PROGRAM MAIN_Fast
VAR
	Router														: FB_Teltonika;
	SystemControl												: FB_SystemControl;
	AcDcCharger													: FB_AcDcCharger;
	ACswitchgear												: FB_ACSwitchgear;
	DCLink														: FB_DCLink;
	HartingIO													: FB_HartingIO;
	NeutralTransformer											: FB_NeutralTransformer;
	Coolingsystem												: FB_Coolingsystem;
	PowerStack													: FB_PowerStack;
	PowerMonitor												: FB_PowerQualityMonitoring;
	InternalPowerSupply											: FB_InternalPowerSupply;
	BMS															: FB_BMS;
	ProtectionSystems											: FB_ProtectionSystems;
	Enclosure													: FB_enclosure;
	PLCstate													: FB_PLCState;
	Peakshavebox												: FB_peakshavebox;
	GenComm														: FB_GenComm;				
END_VAR

VAR // structures containing all system control/monitoring vars and are exchanged with other task.
	{ attribute 'TcHmiSymbol.Hide' }
	monitor						: ST_System_Monitor;
	{ attribute 'TcHmiSymbol.Hide' }
	control						: REFERENCE TO ST_System_Control;

	fb_WritePersistentData		: WritePersistentData;
END_VAR

VAR
	//Reset function
	b_ResetManual			: BOOL;
	ton_EMstopTimeOut		: TON := (PT:= T#30S);
	w_MethodFbs				: WORD;
	tp_ResetDuration		: TP := (PT:= T#2S);
	ton_ForceShutdown		: ton := (PT := T#10S);
	ton_shutdownDelay		: ton := (PT := T#3S);
	b_shutdownInitiated		: BOOL;
	ton_NUCshutdownDelay	: ton := (PT := T#20S);
	
	//Method feedbacks
	EMstopFb				: BYTE;		
	b_EMstopCompleted		: BOOL;
	b_shutdownCompleted		: BOOL;
	b_MethodStartFB			: BOOL;
	r_trigInitialReset		: R_TRIG;
END_VAR

control REF= MAIN_Slow.control;

WearLogging();
SetConfig();
SetSystemMonitorControlvars();

IF __ISVALIDREF(control) AND InitMachine() THEN
	PLCstate();
	
	Safety(b_extEmstopTrigger := SystemControl.toSystem.control.b_EMStop,
		b_enable := GVL.b_SystemReady
		);
		Safety.EDMSignals.b_NetcontactorEDM := Powerstack.b_NetcontEDM;
		Safety.EDMSignals.b_MccbMasterEDM:= Powerstack.b_MasterMccbEDM;
		Safety.EDMSignals.b_MccbSlaveEDM:= Powerstack.b_SlaveMccbEDM;
		
	//call FB
	
	PowerStack(
			e_ACRotationStateExt			:= powermonitor.get.OutputField.e_ACrotationStatus,
			r_PLossInternal					:= 0,
			r_QLossInternal					:= 0,
			st_params						:= settings.MachineParams.Powerstack,
			st_service						:= service.Powerstack,
			st_calibration 					:= settings.Calibration.Powerstack,
			set								:= SystemControl.toSystem.Powerstack,
			b_transportMode					:= systemcontrol.toSystem.b_TransportMode,
			b_DoublePowermodule				:= settings.Configuration.b_DoublePowerModule,
			b_BatteryDCReady				:= BMS.PowerStatus = eHVDC_Powerstatus.ON,
			r_BatteryDCvoltage				:= BMS.get.MBMU.BatteryStatus.r_SystemVoltage,
			b_RotationswitchEnable			:= settings.Configuration.b_AutomaticACrotation,
			b_ExtgridCodeTrip				:= Powermonitor.get.OutputField.r_CurrentUnbalance > settings.GridParams.r_CurrentUnbalanceLimit AND Powermonitor.get.OutputField.ar_Current[0] > 20 AND NOT settings.Configuration.b_NeutralTransformer,
			b_EnableFan						:= coolingsystem.b_FanPowerstackEnable,
			b_OutputConnected				:= ACswitchgear.get.b_OutputMCCBfb,
			b_InputConnected				:= ACswitchgear.get.b_inputMCCBfb,// AND ACswitchgear.get.b_InputContactorfb
			b_InternalACRequired			:= InternalPowerSupply.b_PowerStackACRequired
		);

	PowerMonitor(
		b_enable:= TRUE,
		powerstackGet := powerstack.get,
		b_TNModeActive:= Monitor.protections.Insulation.e_EarthingSystemDetected <> eEarthingsystems.IT,
		b_thirdOutputfieldAvailable := settings.Configuration.b_ThirdOutputConnection,
		b_NeutralTransformerAvailable := settings.Configuration.b_NeutralTransformer,
		b_InputFieldsAvailable := settings.Configuration.b_ACInputConnection
		);
	
	InternalPowerSupply(
			st_PowerstackDemandSupply 	:= Powerstack.st_InternalPsuSupplyRequest, 
			st_CoolingDemandSupply 		:= Coolingsystem.IPSRequest,
			st_ACDCchargerDemandSupply 	:= ACDCCharger.IPSRequest,
			st_DCBusDemandSupply		:=	dclink.st_PowerDemand,
			b_BusbarACAvailable := powerstack.get.b_ACdetected,
			st_params:=Settings.MachineParams.Interpowersupply,
			e_BMSPowerState := BMS.PowerStatus,
			b_ConditioningOnBatteryAllowed := BMS.b_InternalHVDCAllowed
		);

	BMS(
		st_params 		:= settings.MachineParams.BMS,
		st_service		:= service.BMS,
		b_HVDCEnable	:= Internalpowersupply.b_HVDC_Enable,
		set 			:= Systemcontrol.toSystem.BMS,
		by_NoOfStrings	:= Settings.Configuration.by_NoBatteryStrings
	);	

	Enclosure(st_params := Settings.MachineParams.Enclosure, set := SystemControl.toSystem.Enclosure);
		Enclosure.ledstrip.SetMachineStatus(
			b_Error := GVL.b_QuickshutdownActive OR GVL.b_EmergencyShutdownActive OR GVL.b_NormalShutdownActive,
			b_warning := GVL.b_WarningActive,
			b_attention := NOT BMS.get.BatteryInfo.b_chargingAllowed OR NOT BMS.get.BatteryInfo.b_dischargingAllowed,
			b_Normal := BMS.PowerStatus = eHVDC_powerstatus.ON,
			b_off :=  Monitor.system.e_State = eSystemState.Transport,
			r_Soc := BMS.get.BatteryInfo.r_SOCScaled,
			r_DCcurrent := Powerstack.get.r_DCcurrent);

	CoolingSystem(
		st_params := settings.MachineParams.Coolingsystem,
		InverterConditioningRequirement := powerstack.ConditioningRequirement,
		b_HVDC_Available	:=	InternalPowerSupply.Get.b_HVDCAvailable,
		b_400V_Available  := 	InternalPowerSupply.Get.b_400VACAvailable,
		
// 		by_PSsetCooling:= powerstack.by_CoolingControl,
// 		b_InverterRunning:= powerstack.get.b_InverterRunning,
// 		r_InverterLoad := powerstack.get.r_LoadPercent,
// 		b_24v_Available := internalpowersupply.Get.b_24VdcAvailable,
// 		b_400v_Available := internalpowersupply.Get.b_400VACAvailable,
// 		e_400vSupplySource := internalpowersupply.Get.e_400VSupplySource,
// 		r_BMSAverageBattTemp := BMS.get.BatteryInfo.ar_CellTemperature[eSubvalues.Average],
// 		r_BMSMaxBattTemp := BMS.get.BatteryInfo.ar_CellTemperature[eSubvalues.Maximum],
// 		b_DehumStart := systemcontrol.toSystem.control.b_startDeHum,
// 		r_enclosureHumidity := enclosure.get.climate.r_Humidity,
// 		r_enclosureTemperature := enclosure.get.climate.r_Temperature,
// 		r_InverterTemp := Powerstack.get.PowermoduleMaster.r_TemperatureInverter,
// 		b_ConditioningOnBatteryAllowed := BMS.b_InternalHVDCAllowed
		);
		
	
	NeutralTransformer(
		b_enable:= settings.Configuration.b_NeutralTransformer,
		r_currentN := Powermonitor.get.inverter.ar_Current[phases.N],
		r_linevoltage := powermonitor.get.OutputField.ar_LineVoltage[Phases.AVG],
		r_voltageUnbalance := Powermonitor.get.Outputfield.r_VoltageUnbalance,
		b_NetcontactorFB := Powerstack.get.Netcontactor.b_NetConFb,
		st_params := settings.MachineParams.NeutralTransformer
		);
	
		
	ProtectionSystems(
		st_params := settings.MachineParams.Protections,
		powermonitor := Powermonitor.get,
		b_batteryAlarm := BMS.get.Events.b_OVER_TEMP_ALARM
	);
		ProtectionSystems.ToInsuMon.b_MccbfbMaster := Powerstack.get.PowermoduleMaster.b_MccbFb;
		ProtectionSystems.ToInsuMon.b_MccbfbSlave := Powerstack.get.PowermoduleSlave.b_MccbFb;
		ProtectionSystems.ToInsuMon.b_NetContFB := Powerstack.get.Netcontactor.b_NetConFb;
		ProtectionSystems.ToInsuMon.b_ACdetected := Powerstack.get.b_ACdetected;
		ProtectionSystems.ToInsuMon.b_PENlinkFB := AcSwitchgear.get.b_PENlinkfb;
		ProtectionSystems.set := systemcontrol.toSystem.Protections;
		
	ACswitchgear(
		b_inputAvailable:= settings.Configuration.b_ACInputConnection,
		b_NeutralTransformerAvailable := settings.Configuration.b_NeutralTransformer, 
		b_MCCBinputShuntTrip := protectionsystems.get.OvercurrentProtection.b_InputAlarm,
		b_MCCBOutputShuntTrip:= protectionsystems.get.overcurrentprotection.b_OutputAlarm,
		b_TransportMode := Monitor.system.e_State = eSystemState.Transport,
		set := Systemcontrol.toSystem.ACSwitchgear,
		st_params := settings.MachineParams.ACswitchgear,
		);
		
	AcDcCharger(
		st_service := service.ACDCCharger,
		st_params := settings.MachineParams.ACDCCharger,
		enable:= Settings.Configuration.b_DcCharger,
		set := systemcontrol.tosystem.AcDcCharger,(*BMS := BMS.get.BatteryInfo,*) 
		r_Soc := BMS.get.BatteryInfo.r_SOCScaled, 
		r_SystemVoltage := BMS.get.BatteryInfo.r_SystemVoltage,
		r_SystemCurrent := BMS.get.BatteryInfo.r_SystemCurrent,
		r_MaxChargeCurrent := BMS.get.BatteryInfo.r_MaxChargeCurrentAllowed,
		b_BatteryOn := (BMS.get.BatteryInfo.e_BMS_PowerOnStatus = ePowerOnSTatus.On), 
		b_BatteryFullyCharged := (BMS.get.BatteryInfo.e_BMS_Status = eBMS_status.FullCharge)
		);
	
	DcLink(
		st_params := settings.MachineParams.DC,
		r_InvCurrentDC := Powerstack.get.r_DCcurrent,
		r_battCurrent := BMS.get.BatteryInfo.r_SystemCurrent,
		r_DCbusVoltage := BMS.get.BatteryInfo.r_SystemVoltage,
		r_BattCCL := BMS.get.BatteryInfo.r_MaxChargeCurrentAllowed,
		r_BattDCL := BMS.get.BatteryInfo.r_MaxDischargeCurrentAllowed,
		b_DCsafetyOK := safety.get.b_SafetyDCOK,
		set := systemcontrol.toSystem.DCLink	
		);
	
	HartingIO(
		st_params := settings.MachineParams.HartingIO,
		set := systemcontrol.toSystem.HartingIO,
		SystemOperating := Powerstack.get.b_StartedState,
		SystemEmStop := Monitor.system.e_State = eSystemState.EMstop,
		);
		
	GenComm(
		st_params := settings.MachineParams.GenComm,
		set := systemcontrol.toSystem.GenComm);
	
	//external measurement box (PSB)	
	Peakshavebox(st_params := settings.MachineParams.PSB,
		b_enable:= settings.Configuration.b_PeakshaverBoxEnable AND Control.SoftSettings.setup.b_PeakshaveBoxEnable);
	PeakshaveBox.set := systemcontrol.toSystem.Peakshavebox;

	
	//Router --> GPS, 4G, SMS etc.
	Router(
		st_service := service.Router,
		s_message := errorhandling.a_SMSEventBuffer, 
		st_params := Settings.MachineParams.Router,
		s_SerialNumber := settings.Properties.s_SerialNumber
	);
	monitor.system.b_SMSnumberConfigured := Router.SetSMSNumber(control.SoftSettings.system.s_SMSnumber);
	monitor.system.b_CustomNameConfigured:= Router.SetDevName(control.SoftSettings.system.s_SystemName);

	//FB with connection from user to system vars
	SystemControl(
		st_params := settings.MachineParams.system,
		st_calibration := settings.Calibration,
		monitor:= monitor, control:= control);
	

//CALL MAIN FUNCTIONS
	Reset(SystemControl.toSystem.control.b_Reset, NOT GVL.b_SystemReady OR settings.MachineParams.system.b_VDLReset);
	MainSFC();
	//System shutdown --> manually or by firesystem
	SystemShutdown(Systemcontrol.toSystem.control.b_SystemShutdown OR ProtectionSystems.b_SystemShutdownCMD);
END_IF

ACTION _aErrorSequence_entry:
SFCReset := TRUE;
END_ACTION

ACTION _aInit_active:
//INIT state
b_EMstopCompleted :=  FALSE;
Monitor.system.e_State:= eSystemState.Init;
END_ACTION

ACTION _aStandBy_active:
Powerstack.Standbycmd();
Internalpowersupply.HVDC_Enable();

IF systemcontrol.toSystem.b_TransportMode THEN
	// IF Coolingsystem.Shutdown() THEN  --> WHAT TO DO WITH THIS IN NEW COOLING MODULE?
		powerstack.Shutdowncmd();
	//END_IF
	AcSwitchgear.set.b_inputContactorOpen := TRUE;
	Monitor.system.e_State:= eSystemState.Transport;
ELSE
	Monitor.system.e_State:= eSystemState.Init;
	IF  coolingsystem.Get.CoolingSystemState = eCoolingSystemState.Circulating OR 
	coolingsystem.Get.CoolingSystemState = eCoolingSystemState.ActiveCooling OR
	coolingsystem.Get.CoolingSystemState = eCoolingSystemState.ActiveHeating THEN
		Monitor.system.e_State:= eSystemState.Conditioning;
	ELSE
		Monitor.system.e_State:= eSystemState.StandBy;
	END_IF
END_IF
END_ACTION

ACTION a_ContinousActions:
ErrorSFC();
END_ACTION

ACTION a_EmergencyShutdown_active:
SFCReset := TRUE;
b_EMstopCompleted := EMStop();
Monitor.system.e_State := eSystemState.EMstop;
InternalPowersupply.HVDC_disable();
END_ACTION

ACTION a_ErrorSequence_active:
// SFC IDENTIFICATION
Powerstack.Shutdowncmd();
Reset(FALSE, systemcontrol.toSystem.control.b_Reset);

IF GVL.b_EmergencyShutdownActive THEN
	InternalPowersupply.HVDC_disable();
	Monitor.system.e_State := eSystemState.EMstop;
END_IF
END_ACTION

ACTION a_ErrorSequence_exit:
//RELEASE MAINSEQUENCE AFTER ALL ERROR ARE CLEARED
Reset(FALSE, FALSE);
SFCReset := FALSE;
END_ACTION

METHOD PUBLIC CheckDCcurrent : BOOL
VAR_INPUT
	r_in			: REAL;
END_VAR
//checkcurrent is below limit.
CheckDCcurrent := (BMS.get.BatteryInfo.r_SystemCurrent < r_in AND powerstack.get.r_DCcurrent < r_in);
END_METHOD

METHOD EMstop : BOOL

VAR
	EMstopDone	: BOOL;
END_VAR
//EMstopDone := Powerstack.EMstop() AND 
//	Coolingsystem.EMSTOP() AND 
//	Internalpowersupply.EMstop() AND 
//	BMS.EMSTOP() AND 
//	systemcontrol.EMstop();
	
EMstopFb.0 := Powerstack.EMstop();
EMstopFb.1 := Coolingsystem.EMSTOP();
EMstopFb.2 := Internalpowersupply.EMstop();
EMstopFb.3 := BMS.EMSTOP();
EMstopFb.4 := systemcontrol.EMstop();
EMstopFb.5 := ACDCCharger.EMSTOP();;
EMstopFb.6 := TRUE;
EMstopFb.7 := TRUE;

EMstopDone:= EMstopFb = 255;

ton_EMstopTimeOut(IN:= NOT EMstopDone);
EMstop := EMstopDone; //OR ton_EMstopTimeOut.Q;

IF EMstopDone THEN
	EMstopFb := 0;
END_IF

//IF ton_EMstopTimeOut.Q THEN
//	InternalPowersupply.SystemShutdown(FALSE);
//END_IF
END_METHOD

ACTION ErrorSFC:
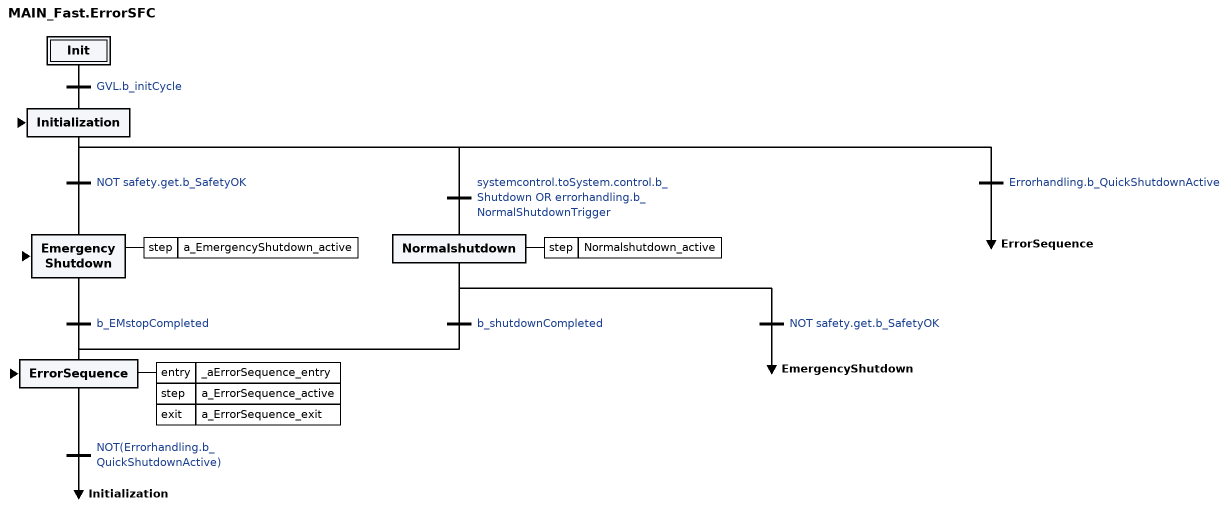
INITIAL_STEP Init:
END_STEP
TRANSITION FROM Init TO Initialization
    := GVL.b_initCycle;
END_TRANSITION
STEP Initialization:
END_STEP
TRANSITION FROM Initialization TO EmergencyShutdown
    := NOT safety.get.b_SafetyOK;
END_TRANSITION
STEP EmergencyShutdown:
    a_EmergencyShutdown_active(N);  // step action
END_STEP
TRANSITION FROM EmergencyShutdown TO ErrorSequence
    := b_EMstopCompleted;
END_TRANSITION
TRANSITION FROM Initialization TO Normalshutdown
    := systemcontrol.toSystem.control.b_Shutdown OR errorhandling.b_NormalShutdownTrigger;
END_TRANSITION
STEP Normalshutdown:
    Normalshutdown_active(N);  // step action
END_STEP
TRANSITION FROM Normalshutdown TO ErrorSequence
    := b_shutdownCompleted;
END_TRANSITION
TRANSITION FROM Normalshutdown TO EmergencyShutdown
    := NOT safety.get.b_SafetyOK;
END_TRANSITION
TRANSITION FROM Initialization TO ErrorSequence
    := Errorhandling.b_QuickShutdownActive;
END_TRANSITION
STEP ErrorSequence:  // min time T#5s
    _aErrorSequence_entry(P1);  // entry action
    a_ErrorSequence_active(N);  // step action
    a_ErrorSequence_exit(P0);  // exit action
END_STEP
TRANSITION FROM ErrorSequence TO Initialization
    := NOT(Errorhandling.b_QuickShutdownActive);
END_TRANSITION
// branch label Branch1_ErrorSFC
// branch label Branch0_ErrorSFC
END_ACTION

ACTION IdleOperation_active:
IF powerstack.stopcmd() THEN
	Monitor.system.e_State := eSystemState.Stopped;
END_IF
END_ACTION

ACTION InitializeMachine_active:

END_ACTION

METHOD PRIVATE InitMachine : Bool
VAR_INPUT
END_VAR
//Calls all available init methods of other function blocks.
//After all inits have returned true, the method returns true and main_fast operation can continue

InitMachine := TRUE;//BMS.init() AND FB.init();
END_METHOD

ACTION MainSFC:
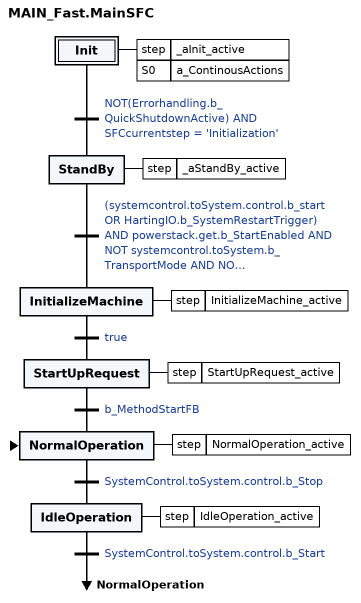
INITIAL_STEP Init:
    _aInit_active(N);  // step action
    a_ContinousActions(S0);
END_STEP
TRANSITION FROM Init TO StandBy
    := NOT(Errorhandling.b_QuickShutdownActive) AND SFCcurrentstep = 'Initialization';
END_TRANSITION
STEP StandBy:
    _aStandBy_active(N);  // step action
END_STEP
TRANSITION FROM StandBy TO InitializeMachine
    := (systemcontrol.toSystem.control.b_start OR HartingIO.b_SystemRestartTrigger) AND powerstack.get.b_StartEnabled AND NOT systemcontrol.toSystem.b_TransportMode AND NOT GVL.b_NormalShutdownActive;
END_TRANSITION
STEP InitializeMachine:
    InitializeMachine_active(N);  // step action
END_STEP
TRANSITION FROM InitializeMachine TO StartUpRequest
    := true;
END_TRANSITION
STEP StartUpRequest:
    StartUpRequest_active(N);  // step action
END_STEP
TRANSITION FROM StartUpRequest TO NormalOperation
    := b_MethodStartFB;
END_TRANSITION
STEP NormalOperation:
    NormalOperation_active(N);  // step action
END_STEP
TRANSITION FROM NormalOperation TO IdleOperation
    := SystemControl.toSystem.control.b_Stop;
END_TRANSITION
STEP IdleOperation:
    IdleOperation_active(N);  // step action
END_STEP
TRANSITION FROM IdleOperation TO NormalOperation
    := SystemControl.toSystem.control.b_Start;
END_TRANSITION
END_ACTION

ACTION NormalOperation_active:
powerstack.startcmd();

IF powerstack.get.e_State = eStatusPowerstack.running THEN
	IF NOT bms.get.BatteryInfo.b_chargingAllowed THEN
		Monitor.system.e_State := eSystemState.Discharging_Only;
	ELSIF NOT bms.get.BatteryInfo.b_DischargingAllowed THEN
		Monitor.system.e_State := eSystemState.Charging_Only;
	ELSE
		Monitor.system.e_State := eSystemState.Running;
	END_IF
ELSE
	IF powerstack.get.e_State = eStatusPowerstack.idle OR powerstack.get.e_State = eStatusPowerstack.GridCodeStop THEN
		Monitor.system.e_State := eSystemState.Stopped;	
	ELSE
		Monitor.system.e_State := eSystemState.Starting;	
	END_IF	
END_IF
END_ACTION

ACTION Normalshutdown_active:
SFCReset := TRUE;
b_shutdownCompleted := Powerstack.Shutdowncmd();
Monitor.system.e_State := eSystemState.shutdown;
END_ACTION

METHOD PUBLIC Reset : BOOL
VAR_INPUT
	b_reset	: BOOL;
	b_force : BOOL;
END_VAR
tp_ResetDuration(IN := b_reset OR b_Force);

//reinitiliaze reset statuss if reset is retriggered
IF tp_resetDuration.Q = FALSE THEN
	w_MethodFbs := 0;
END_IF


//Everything that is not automatically reset
IF tp_ResetDuration.Q AND w_MethodFbs <> 16#FF THEN
	monitor.system.e_State := eSystemState.Reset;
	
	IF NOT w_MethodFbs.0 AND b_force THEN w_MethodFbs.0 := Safety.Reset(TRUE); END_IF
	IF NOT w_MethodFbs.1 THEN w_MethodFbs.1 := InternalPowerSupply.Reset(); END_IF
	IF NOT w_MethodFbs.2 THEN w_MethodFbs.2 := Powerstack.Reset(); END_IF
	IF NOT w_MethodFbs.3 THEN w_MethodFbs.3 := protectionSystems.Reset(); END_IF
	IF NOT w_MethodFbs.4 THEN w_MethodFbs.4 := Powermonitor.Reset(); END_IF 
	IF NOT w_MethodFbs.5 THEN w_MethodFbs.5 := BMS.Reset(); END_IF 
	IF NOT w_MethodFbs.6 THEN w_MethodFbs.6 := Neutraltransformer.Reset(); END_IF
	IF NOT w_MethodFbs.7 THEN w_MethodFbs.7 := Coolingsystem.Reset(); END_IF
	IF NOT w_MethodFbs.8 THEN w_MethodFbs.8 := Router.Reset(); END_IF
	IF NOT w_MethodFbs.9 THEN w_MethodFbs.9	:= systemcontrol.Reset(); END_IF
	IF NOT w_MethodFbs.10 THEN w_MethodFbs.10:= ACDCCharger.Reset(); END_IF
	IF NOT w_MethodFbs.11 THEN w_MethodFbs.11:= TRUE; END_IF
	IF NOT w_MethodFbs.12 THEN w_MethodFbs.12:= TRUE; END_IF
	IF NOT w_MethodFbs.13 THEN w_MethodFbs.13:= TRUE; END_IF
	IF NOT w_MethodFbs.14 THEN w_MethodFbs.14:= TRUE; END_IF
	IF NOT w_MethodFbs.15 THEN w_MethodFbs.15:= TRUE; END_IF
END_IF

//Everything that is automatically reset one in error state
Reset := w_MethodFbs = 255;
END_METHOD

ACTION SetConfig:
{IF defined (ePU10_360_N_DC_IO_PSB)}
	settings.Configuration.b_PeakshaverBoxEnable 	:= TRUE;
	settings.Configuration.b_DCbuscoupling 			:= FALSE; //TRUE;
	settings.Configuration.b_NeutralTransformer		:= TRUE;
	settings.Configuration.b_ACInputConnection		:= TRUE;
	settings.Properties.s_ConfigurationCode 		:= 'ePU10_360_N_DC_IO_PSB';
{END_IF}

{IF defined (ePU10_360_N_IO_PSB)}
	settings.Properties.s_ConfigurationCode 		:= 'ePU10_360_N_IO_PSB';
	settings.Configuration.b_ACInputConnection		:= TRUE;
	settings.Configuration.b_NeutralTransformer		:= TRUE;
	settings.Configuration.b_PeakshaverBoxEnable 	:= TRUE;
{END_IF}

{IF defined (ePU10_360_N_IO)}
	settings.Properties.s_ConfigurationCode 		:= 'ePU10_360_N_IO';
	settings.Configuration.b_ACInputConnection		:= TRUE;
	settings.Configuration.b_NeutralTransformer		:= TRUE;
{END_IF}

{IF defined (ePU10_368_3P_O_PSB)}
	settings.Properties.s_ConfigurationCode 		:= 'ePU10_368_3P_O_PSB';
	settings.Configuration.b_PeakshaverBoxEnable 	:= TRUE;
{END_IF}

{IF defined (ePU10_360_3P_O)}
	settings.Properties.s_ConfigurationCode 		:= 'ePU10_360_3P_O';
{END_IF}

IF enclosure.get.ledstrip.BeckhoffLed AND FIND(settings.Properties.s_ConfigurationCode,'_BL') = 0 THEN
	settings.Properties.s_ConfigurationCode := CONCAT(settings.Properties.s_ConfigurationCode, '_BL');
END_IF

settings.Properties.by_SWverMajor	:=	1;	
settings.Properties.by_SWverMinor	:=	6;	
settings.Properties.by_SWverPatch	:=	1;	
settings.Properties.by_SWverBuild	:=	1;	

//Set properties
settings.Properties.s_SWversionNumber				:= 	concat('V', TO_STRING(settings.Properties.by_SWverMajor));
settings.Properties.s_SWversionNumber				:=	concat(settings.Properties.s_SWversionNumber, '.');
settings.Properties.s_SWversionNumber				:= 	concat(settings.Properties.s_SWversionNumber, TO_STRING(settings.Properties.by_SWverMinor));
settings.Properties.s_SWversionNumber				:=	concat(settings.Properties.s_SWversionNumber, '.');
settings.Properties.s_SWversionNumber				:= 	concat(settings.Properties.s_SWversionNumber, TO_STRING(settings.Properties.by_SWverPatch));
IF settings.Properties.by_SWverBuild > 0 THEN
	settings.Properties.s_SWversionNumber				:=	concat(settings.Properties.s_SWversionNumber, '_');
	settings.Properties.s_SWversionNumber				:= 	concat(settings.Properties.s_SWversionNumber, TO_STRING(settings.Properties.by_SWverBuild));
END_IF
	
settings.Properties.r_RatedEnergyCapacity 			:= BMS.get.BatteryInfo.r_ratedEnergyCapacity;
settings.Properties.r_RatedActivePower 				:= MIN(BMS.get.BatteryInfo.r_ratedPower, powerstack.get.r_ratedPower);
settings.Properties.r_RatedApparentPower			:= TO_INT(powerstack.get.r_RatedCurrent * 400 * 1.73 / 1000);
settings.Properties.r_Ratedcurrent 					:= powerstack.get.r_RatedCurrent;
settings.Properties.r_ratedCurrentInput				:= SEL(settings.Configuration.b_ACInputConnection, 0, 700);
settings.Properties.r_ratedCurrentOutput			:= SEL(settings.Configuration.b_ThirdOutputConnection, 800, 1200);


CASE settings.Configuration.by_NoBatteryStrings OF
	2: settings.Properties.s_Weight					:= '7000 kg';
	3: settings.Properties.s_Weight					:= '8500 kg';
	4: settings.Properties.s_Weight					:= '9500 kg';
END_CASE
END_ACTION

ACTION SetSystemMonitorControlvars:
//First bind references
Monitor.safety := Safety.get;
Monitor.powerstack REF= Powerstack.get;
Monitor.AcDcCharger REF= AcDcCharger.get;
Monitor.powermonitor REF= Powermonitor.get;
Monitor.neutraltransformer REF= neutraltransformer.get;
Monitor.protections REF= ProtectionSystems.get;
Monitor.battery REF= BMS.get;
Monitor.ACswitchgear REF= ACswitchgear.get;
Monitor.DCLink REF= DCLink.get;
Monitor.peakshavebox REF= Peakshavebox.get;
Monitor.enclosure REF= Enclosure.get;
Monitor.internalpsu REF= Internalpowersupply.Get;
Monitor.PLC REF= PLCstate.get;
Monitor.Cooling REF= coolingsystem.Get;
Monitor.Router REF= Router.Get;
Monitor.Generator REF= Gencomm.Get;
Monitor.HartingIO REF= HartingIO.Get;
END_ACTION

ACTION StartUpRequest_active:
b_MethodStartFB	:= Powerstack.Startcmd();
Monitor.system.e_State:= eSystemState.Starting;
END_ACTION

METHOD SystemShutdown : BOOL
VAR_INPUT
	b_execute			: BOOL;
END_VAR
//write persisten data
fb_WritePersistentData(NETID := '', PORT:= 851, START:=b_execute,  TMOUT := T#5S);

//set force shutdown timer
ton_ForceShutdown(IN:= b_execute);
ton_shutdownDelay(IN:= b_execute);

IF ton_shutdownDelay.Q THEN
	b_shutdownInitiated := TRUE;
END_IF

//Everything that is not automatically reset
IF b_shutdownInitiated THEN
	settings.Save := TRUE;
	Monitor.system.e_State := eSystemState.shutdown;
	IF NOT w_MethodFbs.0 THEN w_MethodFbs.0 := Powerstack.Shutdowncmd(); END_IF	
	IF NOT w_MethodFbs.1 THEN w_MethodFbs.1 := SystemControl.shutdown(); END_IF
	IF NOT w_MethodFbs.2 THEN w_MethodFbs.2 := CoolingSystem.shutdown(); END_IF;
	w_MethodFbs.3 := TRUE;	
	w_MethodFbs.4 := TRUE; 
	w_MethodFbs.5 := TRUE; 
	w_MethodFbs.6 := TRUE; 
	w_MethodFbs.7 := TRUE;
ELSE
	w_MethodFbs := 0;
END_IF

IF w_MethodFbs = 255 OR ton_ForceShutdown.Q THEN
	settings.Save := FALSE;
	MqttComOpenRemote.shutdown();
	ton_NUCshutdownDelay(IN:=TRUE);
	IF ton_NUCshutdownDelay.Q THEN
		Monitor.system.e_State := eSystemState.off;
		InternalPowerSupply.SystemShutdown(timedshutdown := FALSE);
		b_shutdownInitiated := FALSE;
	END_IF
END_IF
END_METHOD

END_PROGRAM

(* stored: Version 1.1.0.1, ProductVersion 3.1.4026.18
   POU MAIN_Fast: Id {c3f9cfcc-0865-4c2f-9fe3-3cc41bfe2f16}, SpecialFunc None
   Folder SFC: Id {e3e26b5f-f1e8-47e6-a64d-4aa0da400882}
   Action _aErrorSequence_entry: Id {1b93d4fa-78ca-47ae-85b4-4ece75f01b15}
   Action _aInit_active: Id {effe53df-6a9d-4897-a064-92b16ed612db}
   Action _aStandBy_active: Id {8b351738-c15a-40bc-af25-8570c9331b8e}
   Action a_ContinousActions: Id {05c6989e-311b-4791-aca1-bb295fcfd946}
   Action a_EmergencyShutdown_active: Id {b86c67cf-82ba-4cb1-ad85-40515fa44753}
   Action a_ErrorSequence_active: Id {8c0a0457-7263-4e49-add3-136bfbc6663a}
   Action a_ErrorSequence_exit: Id {edde1199-4f99-4b0f-b15c-c5f29e8fc03b}
   Method CheckDCcurrent: Id {894e27fd-7344-41a9-87ad-52eadf33d1ca}
   Method EMstop: Id {d110c828-9456-4fbe-bfdd-d6633d4c6709}
   Action ErrorSFC: Id {0329997e-c4aa-4da2-8bb2-5babd452e15d}
   Action IdleOperation_active: Id {99fb1725-e090-4871-89ff-b9ea45a04197}
   Action InitializeMachine_active: Id {40796f25-d82c-4764-a6db-87f7967ace80}
   Method InitMachine: Id {7cbfe594-92e9-485f-b7c4-e39dadfdb8ef}
   Action MainSFC: Id {4d748394-499c-4b67-8b1d-40f0b63a6d02}
   Action NormalOperation_active: Id {56d2521e-6356-496d-8aa8-0d2424f5790f}
   Action Normalshutdown_active: Id {4d0315ce-a511-4ec5-8ddf-10cce2cbe602}
   Method Reset: Id {7a48efb2-2c09-45a8-bebd-e7f87f31865d}
   Action SetConfig: Id {d70e48b1-da73-45d4-a3da-134966cb20f4}
   Action SetSystemMonitorControlvars: Id {ee1ac32e-4a18-4b7d-a1ed-f24635a6285c}
   Action StartUpRequest_active: Id {090a0f6e-3020-4e2f-b065-9b9ede2298d7}
   Method SystemShutdown: Id {5d76c95d-5fda-40b0-8826-8b775359b161} *)
